Fanuc TP program (LS listing): tool_offset.ls

/PROG  TOOL_OFFSET
/ATTR
OWNER		= MNEDITOR;
COMMENT		= "";
PROG_SIZE	= 199;
CREATE		= DATE 21-02-09  TIME 06:04:28;
MODIFIED	= DATE 21-02-21  TIME 07:47:06;
FILE_NAME	= ;
VERSION		= 0;
LINE_COUNT	= 2;
MEMORY_SIZE	= 563;
PROTECT		= READ_WRITE;
TCD:  STACK_SIZE	= 0,
      TASK_PRIORITY	= 50,
      TIME_SLICE	= 0,
      BUSY_LAMP_OFF	= 0,
      ABORT_REQUEST	= 0,
      PAUSE_REQUEST	= 0;
DEFAULT_GROUP	= 1,*,*,*,*;
CONTROL_CODE	= 00000000 00000000;
/APPL

AUTO_SINGULARITY_HEADER;
  ENABLE_SINGULARITY_AVOIDANCE   : TRUE;
/MN
   1:  PR[9]=LPOS    ;
   2:L PR[9] 50mm/sec FINE Tool_Offset,PR[10]    ;
/POS
/END
